// TwinCAT 3 PLC project Untitled1
// ProgramVersion: 3.1.4020.10
// libraries:
//   Tc2_Standard, * (Beckhoff Automation GmbH)
//   Tc2_System, * (Beckhoff Automation GmbH)
//   Tc2_TcpIp, * (Beckhoff Automation GmbH)
//   Tc3_Module, * (Beckhoff Automation GmbH)
// project tree:
//   DUTs/ E_ClientSteps.TcDUT, E_DataExchaSteps.TcDUT, E_ServerSteps.TcDUT (not stored)
//   GVLs/ GVL.TcGVL (not stored)
//   / PlcTask.TcTTO
//   POUs/ MAIN.TcPOU (not stored)
// real-time tasks:
//   TASK PlcTask: cycle T#10ms, priority 20, ADS port 350
// I/O:
//   DEVICE Device 1 (EtherCAT), AmsNetId 169.254.245.7.2.1
//     Term 1 (EK1200) [EK1200-5000 EtherCAT Power supply (2A E-Bus)]
//       Term 2 (EL2088) [EL2088 8Ch. Dig. Output 24V, 0.5A, switching to negative]
//       Term 3 (EL9011) [EL9011 End Terminal]
//   DEVICE Device 4 (COM Port)
// variable links:
//   Untitled1/Untitled1 Instance <-> Device 1 (EtherCAT)/Term 1 (EK1200)/Term 2 (EL2088)
//     PlcTask Outputs/MAIN.bOUt1 <-> Channel 1/Output
//     PlcTask Outputs/MAIN.bOut2 <-> Channel 2/Output

CONFIGURATION Untitled1
    RESOURCE PLC ON TwinCAT3
        TASK PlcTask(INTERVAL := T#10ms, PRIORITY := 20);
        PROGRAM MAIN WITH PlcTask : MAIN;
    END_RESOURCE
END_CONFIGURATION

// ---- DUTs/E_ClientSteps.TcDUT
TYPE E_ClientSteps :
(
	CLIENT_STATE_IDLE,
	CLIENT_STATE_CONNECT_START,
	CLIENT_STATE_CONNECT_WAIT,
	CLIENT_STATE_DATAEXCHA_START,
	CLIENT_STATE_DATAEXCHA_WAIT,
	CLIENT_STATE_CLOSE_START,
	CLIENT_STATE_CLOSE_WAIT,
	CLIENT_STATE_ERROR
);
END_TYPE

// ---- DUTs/E_DataExchaSteps.TcDUT
TYPE E_DataExchaSteps :
(
	DATAEXCHA_STATE_IDLE,
	DATAEXCHA_STATE_SEND_START,
	DATAEXCHA_STATE_SEND_WAIT,
	DATAEXCHA_STATE_RECEIVE_START,
	DATAEXCHA_STATE_RECEIVE_WAIT,
	DATAEXCHA_STATE_ERROR
);
END_TYPE
